{attribute 'GeneratedUsingTerminal: KL8001-0002'}
{attribute addProperty BoxType "KL8001-0002"}
{attribute addProperty Id "Channel_1AT %Q*Channel_2F3145090"}
{attribute addProperty CRC "2006552799"}
{attribute addProperty Size "0"}
TYPE KL_779990DF :
STRUCT
	{attribute addProperty Name "Channel_1"}
	Channel_1 : Channel_2F314509;
END_STRUCT
END_TYPE

(* stored: Version 1.2.0.0, ProductVersion 3.1.4024.9
   DUT KL_779990DF: Id {1b0f0ae2-d10a-4eac-a028-033e9c0f7db3} *)
